(* IEC 61131-3 sources: ae-simplified-sorting-machine/AX/src/packagingSortingMachine, 4 files *)

(* ---- BoxGenerator.st ---- *)
USING SortingMachine;
USING Siemens.Simatic.Crypto;

NAMESPACE SortingMachine

    /// Configuration structure for BoxGenerator
    TYPE
        BoxGeneratorConfig : STRUCT
            /// Default width for generated boxes
            defaultWidth : INT := 50;
            /// Default start position for generated boxes
            defaultStartPosition : INT := 0;
            /// Color code for X-type boxes (typically green)
            colorX : WSTRING := "0xFF21BA84";
            /// Color code for Y-type boxes (typically yellow)
            colorY : WSTRING := "0xFFE8C100";
            /// Starting ID for box numbering (auto-incremented)
            startingId : UINT := UINT#1;
            /// Enable automatic ID increment
            autoIncrementId : BOOL := TRUE;
        END_STRUCT;

    END_TYPE

    /// Box generator class for creating different types of boxes
    /// Provides methods to generate X-type, Y-type, and random boxes with configurable properties
    CLASS PUBLIC BoxGenerator
        VAR PRIVATE
            /// Configuration for the box generator
            _config : BoxGeneratorConfig;
            /// Current ID counter for generated boxes
            _currentId : UINT := UINT#1;
        END_VAR

        /// Constructor to configure the box generator
        METHOD PUBLIC CONSTRUCTOR
            VAR_INPUT
                /// Configuration structure with default values and color settings
                config : BoxGeneratorConfig;
            END_VAR
            _config := config;
            _currentId := _config.startingId;
        END_METHOD

        /// Constructor with individual parameters for convenience
        METHOD PUBLIC CONSTRUCTOR
            VAR_INPUT
                /// Default width for all generated boxes
                defaultWidth : INT;
                /// Default start position for all generated boxes
                defaultStartPosition : INT;
                /// Color code for X-type boxes
                colorX : WSTRING;
                /// Color code for Y-type boxes
                colorY : WSTRING;
                /// Starting ID for box numbering
                startingId : UINT := UINT#1;
            END_VAR
            _config.defaultWidth := defaultWidth;
            _config.defaultStartPosition := defaultStartPosition;
            _config.colorX := colorX;
            _config.colorY := colorY;
            _config.startingId := startingId;
            _config.autoIncrementId := TRUE;
            _currentId := startingId;
        END_METHOD

        /// Create a new box
        METHOD PRIVATE CreateBox
            VAR_INPUT
                /// Optional custom ID, if 0 uses auto-increment
                customId : UINT := UINT#0;
                /// Optional custom start position, if 0 uses default
                customStartPos : INT := 0;
                /// Color to use for the box
                customColor : WSTRING;
            END_VAR
            VAR_IN_OUT
                /// New BasicBox instance configured as specified
                newBox : BasicBox;
            END_VAR

            VAR_TEMP
                useId : UINT;
                useStartPos : INT;
            END_VAR

            // Determine ID to use
            IF customId <> UINT#0 THEN
                useId := customId;
            ELSE
                useId := _currentId;
                IF _config.autoIncrementId THEN
                    _currentId := _currentId + UINT#1;
                END_IF;
            END_IF;

            // Determine start position to use
            IF customStartPos <> 0 THEN
                useStartPos := customStartPos;
            ELSE
                useStartPos := _config.defaultStartPosition;
            END_IF;

            newBox.CONSTRUCT(
                id := useId,
                baseColor := customColor,
                width := _config.defaultWidth,
                startPosition := useStartPos
            );
        END_METHOD

        /// Create a new X-type box (typically green)
        METHOD PUBLIC CreateBoxX
            VAR_INPUT
                /// Optional custom ID, if 0 uses auto-increment
                customId : UINT := UINT#0;
                /// Optional custom start position, if 0 uses default
                customStartPos : INT := 0;
            END_VAR
            VAR_IN_OUT
                /// New BasicBox instance configured as X-type
                newBox : BasicBox;
            END_VAR

            THIS.CreateBox(
                customId := customId,
                customStartPos := customStartPos,
                customColor := _config.colorX,
                newBox := newBox);
        END_METHOD

        /// Create a new Y-type box (typically yellow)
        METHOD PUBLIC CreateBoxY
            VAR_INPUT
                /// Optional custom ID, if 0 uses auto-increment
                customId : UINT := UINT#0;
                /// Optional custom width, if 0 uses default (currently unused)
                customWidth : INT := 0;
                /// Optional custom start position, if 0 uses default
                customStartPos : INT := 0;
            END_VAR
            VAR_IN_OUT
                /// New BasicBox instance configured as Y-type
                newBox : BasicBox;
            END_VAR

            THIS.CreateBox(
                customId := customId,
                customStartPos := customStartPos,
                customColor := _config.colorY,
                newBox := newBox);
        END_METHOD

        /// Create a random box (randomly X-type or Y-type)
        METHOD PUBLIC CreateRandomBox
            VAR_INPUT
                /// Optional custom ID, if 0 uses auto-increment
                customId : UINT := UINT#0;
                /// Optional custom start position, if 0 uses default
                customStartPos : INT := 0;
            END_VAR
            VAR_IN_OUT
                /// New BasicBox instance with random type (X or Y)
                newBox : BasicBox;
            END_VAR
            VAR_TEMP
                randomValue : UDINT;
                useColor : WSTRING;
            END_VAR

            // Generate random value using simple linear congruential generator
            randomValue := Random();

            // Determine color based on random value (even = X, odd = Y)
            IF (randomValue MOD UDINT#2) = UDINT#0 THEN
                useColor := _config.colorX;
            ELSE
                useColor := _config.colorY;
            END_IF;

            THIS.CreateBox(
                customId := customId,
                customStartPos := customStartPos,
                customColor := useColor,
                newBox := newBox);
        END_METHOD

        /// Get the current configuration
        METHOD PUBLIC GetConfig : BoxGeneratorConfig
            GetConfig := _config;
        END_METHOD

        /// Update the configuration
        METHOD PUBLIC SetConfig
            VAR_INPUT
                /// New configuration to apply
                config : BoxGeneratorConfig;
            END_VAR
            _config := config;
        END_METHOD

        /// Get the current ID that would be used for the next box
        METHOD PUBLIC GetCurrentId : UINT
            GetCurrentId := _currentId;
        END_METHOD

        /// Set the current ID counter
        METHOD PUBLIC SetCurrentId
            VAR_INPUT
                /// New ID value to use for subsequent boxes
                newId : UINT;
            END_VAR
            _currentId := newId;
        END_METHOD

        /// Reset the ID counter to the starting value
        METHOD PUBLIC ResetIdCounter
            _currentId := _config.startingId;
        END_METHOD
    END_CLASS

END_NAMESPACE

(* ---- IBasicBox.st ---- *)
NAMESPACE SortingMachine

    /// Data structure representing box properties and status
    /// Used for tracking boxes within the sorting machine system
    INTERFACE IBasicBox
        //=============================================================================
        //SIEMENS AG
        //(c)Copyright 2025 All Rights Reserved
        //-----------------------------------------------------------------------------
        //Tested with:   S7-1500 FW V4.0
        //Engineering:   SIMATIC AX Logic Control Engineering
        //Requirements:  none
        //Functionality: Data structure representing box properties and status
        //-----------------------------------------------------------------------------
        //Change log table:
        //Version  Date       Expert in charge                Changes applied
        //01.00.00 28.11.2025 Siemens Industry Online Support First Release
        //=============================================================================

        /// Constructor to be called once and set private variables
        METHOD CONSTRUCT
            VAR_INPUT
                id : UINT;
                baseColor : WSTRING;
                width   : INT;
                startPosition : INT;
            END_VAR
        END_METHOD

        /// Clear all Data from _boxData
        METHOD  ClearData : BOOL
        END_METHOD

        /// Move the Boxe using the inputed increment value
        METHOD  MoveIncrement : INT
            VAR_INPUT
                increment : INT;
            END_VAR
        END_METHOD

        /// Get Box internal Data
        METHOD  GetBoxData : typeBoxData
        END_METHOD
    END_INTERFACE
END_NAMESPACE

(* ---- AutomaticModeCoordinator.st ---- *)
USING SortingMachine;
USING IEC;
USING Siemens.Simatic.Alarming;

NAMESPACE SortingMachine
    /// Function block for coordinating automatic mode operation of the sorting machine
    /// Handles the automatic flow of boxes through conveyor stations and elevator
    /// Manages the sequence: ConveyorStation1 → Elevator → ConveyorStation2/3 based on box properties
    FUNCTION_BLOCK AutomaticModeCoordinator
        //=============================================================================
        //SIEMENS AG
        //(c)Copyright 2025 All Rights Reserved
        //-----------------------------------------------------------------------------
        //Tested with:   S7-1500 FW V4.0
        //Engineering:   SIMATIC AX Logic Control Engineering
        //Requirements:  none
        //Functionality: Automatic mode coordinator for sorting machine
        //-----------------------------------------------------------------------------
        //Change log table:
        //Version  Date       Expert in charge                Changes applied
        //01.00.00 28.11.2025 Siemens Industry Online Support First Release
        //=============================================================================
        VAR_INPUT
            /// Enable automatic mode operation
            enable : BOOL;
            /// Reset the automatic sequence to initial state
            reset : BOOL;
        END_VAR
        VAR_OUTPUT
            /// Automatic mode is active and running
            active : BOOL;
            /// Error occurred during automatic operation
            error : BOOL;
            /// Status code describing current operation
            status : WORD;
            /// Stored boxes after output conveyors
            storedBoxes : typeStorageInterface;
        END_VAR
        VAR_IN_OUT
            /// Reference to input conveyor station
            conveyorStation1 : ConveyorStation;
            /// Reference to elevator station
            elevatorStation : ElevatorBiStateStation;
            /// Reference to upper output conveyor station
            conveyorStation2 : ConveyorStation;
            /// Reference to lower output conveyor station
            conveyorStation3 : ConveyorStation;
            /// Initial box to use for starting the sequence
            initialBox : BasicBox;
        END_VAR
        VAR PRIVATE
            /// Maximum timeout for operations (30 seconds)
            _maxOperationTime : TIME := T#30s;
            /// Scaner simulation timer to continue
            _scanStationTime : TON;
            /// Elevator delay time for the visualization
            _elevatorDelayTime : TON;
            /// Coordinator was previously reset
            _prevReset : BOOL;
            /// Box amount tracker
            _boxAmountTracker : BoxAmountTracker;
            /// S7-1500 program Alarm for Automatic mode coordenator
            {S7.Alarm = NoAck, "Automatic Mode in Error"}
            alarmAutomaticMode : ProgramAlarm;
        END_VAR
        VAR_TEMP
            elevatorPosition : typeElevatorPosition;
        END_VAR
        VAR CONSTANT
            // Scanner simulation time
            SCAN_SIMULATION_TIME : LTIME := LTIME#2S;
            // Elevator Delay simulation time
            ELEVATOR_SIMULATION_TIME : LTIME := LTIME#1S;
        END_VAR
        // Handle reset request
        IF reset AND NOT _prevReset THEN
            error := FALSE;
            _scanStationTime(IN := FALSE);
            _elevatorDelayTime(IN := FALSE);
            status := typeAutomaticModeCoordinatorStatus#STATUS_RESET_COMPLETE;
        END_IF;
        // Update active status
        active := enable AND NOT error;
        _scanStationTime(IN := conveyorStation1.ReadyToRemoveBox(), PT := SCAN_SIMULATION_TIME);
        _elevatorDelayTime(IN := elevatorStation.ReadyToRemoveBox(), PT := ELEVATOR_SIMULATION_TIME);
        // Update previous flags
        _prevReset := reset;
        // Automatic mode alarm
        alarmAutomaticMode(sig := error);
        // Only run if enabled
        IF NOT (enable OR error) THEN
            status := typeAutomaticModeCoordinatorStatus#STATUS_AUTOMATIC_MODE_DISABLED;
            RETURN;
        END_IF;
        // Check for errors in stations and stop if there are errors
        IF conveyorStation1.GetError()
            OR elevatorStation.GetError()
            OR conveyorStation2.GetError()
            OR conveyorStation3.GetError()
            OR error THEN
            error := TRUE;
            status := typeAutomaticModeCoordinatorStatus#ERR_STATION_FAULT;
            RETURN;
        ELSE
            status := typeAutomaticModeCoordinatorStatus#STATUS_NO_CALL;
        END_IF;

        // Automatic handling for each station
        // Conveyor Station 1:
        // Add initial box if needed
        IF initialBox.BoxData.isPresent AND conveyorStation1.ReadyToReciveBox() THEN
            conveyorStation1.AddNewBox(initialBox);
            initialBox.ClearData();
        // Move box from conv1 to elevator if needed
        ELSIF _scanStationTime.Q AND elevatorStation.ReadyToReciveBox() THEN
            elevatorStation.AddNewBox(conveyorStation1.RemoveBox());
        // Move conveyor boxes
        ELSIF NOT conveyorStation1.GetIsMoving() THEN
                conveyorStation1.MoveIncrementForward();
        END_IF;

        // Elevator 1:
        // Move box from elevator to conveyors
        IF _elevatorDelayTime.Q  OR TRUE THEN
            elevatorPosition := elevatorStation.GetElevatorPositionEnum();
            CASE elevatorPosition OF
                typeElevatorPosition#WORK_POS_1, typeElevatorPosition#HOME:
                    // Transfer to lower output conveyor (ConveyorStation3)
                    IF conveyorStation3.ReadyToReciveBox() THEN
                        conveyorStation3.AddNewBox(elevatorStation.RemoveBox());
                    END_IF;
                typeElevatorPosition#WORK_POS_2:
                    // Transfer to upper output conveyor (ConveyorStation2)
                    IF conveyorStation2.ReadyToReciveBox() THEN
                        conveyorStation2.AddNewBox(elevatorStation.RemoveBox());
                    END_IF;
            END_CASE;
        END_IF;

        // Conveyor 2:
        // Remove boxes from output conveyor 2
        IF conveyorStation2.ReadyToRemoveBox() THEN
            conveyorStation2.RemoveBox();
            _boxAmountTracker.addBoxY := TRUE;
        // Continue moving Conveyor
        ELSIF NOT conveyorStation2.GetIsMoving() THEN
            conveyorStation2.MoveIncrementForward();
        END_IF;
        // Conveyor 3:
        // Remove boxes from output conveyor 3
        IF conveyorStation3.ReadyToRemoveBox() THEN
            conveyorStation3.RemoveBox();
            _boxAmountTracker.addBoxX := TRUE;
        // Continue moving Conveyor
        ELSIF NOT conveyorStation3.GetIsMoving() THEN
            conveyorStation3.MoveIncrementForward();
        END_IF;

        // Track box additions
        _boxAmountTracker(
            reset := reset,
            storedBoxes => storedBoxes);
        // Reset add box inputs for next cycle
        _boxAmountTracker.addBoxX := FALSE;
        _boxAmountTracker.addBoxY := FALSE;

    END_FUNCTION_BLOCK
END_NAMESPACE

(* ---- BasicBox.st ---- *)
NAMESPACE SortingMachine
    /// Basic implementation of a Box in the sorting machine
    CLASS PUBLIC BasicBox IMPLEMENTS IBasicBox
        //=============================================================================
        //SIEMENS AG
        //(c)Copyright 2025 All Rights Reserved
        //-----------------------------------------------------------------------------
        //Tested with:   S7-1500 FW V4.0
        //Engineering:   SIMATIC AX Logic Control Engineering
        //Requirements:  none
        //Functionality: Data structure representing box properties and status
        //-----------------------------------------------------------------------------
        //Change log table:
        //Version  Date       Expert in charge                Changes applied
        //01.00.00 28.11.2025 Siemens Industry Online Support First Release
        //=============================================================================
        VAR PUBLIC
            /// Box data with all relevant properties
            BoxData : typeBoxData;
        END_VAR

        /// Constructor to be called once and set variables
        METHOD PUBLIC CONSTRUCT
            VAR_INPUT
                id : UINT;
                baseColor : WSTRING;
                width   : INT;
                startPosition : INT;
            END_VAR
            BoxData.id := id;
            BoxData.baseColor := baseColor;
            BoxData.isPresent := TRUE;
            BoxData.width := width;
            BoxData.posLeft := startPosition;
            ;
        END_METHOD

        /// Constructor to be called once and set variables based on another Box properties
        METHOD PUBLIC CONSTRUCT
            VAR_IN_OUT
                newBox : BasicBox;
            END_VAR
            BoxData := newBox.BoxData;
            ;
        END_METHOD

        /// Constructor to be called once and set variables based on another Box properties
        METHOD PUBLIC CONSTRUCT
            VAR_INPUT
                newBox : typeBoxData;
            END_VAR
            BoxData := newBox;
            ;
        END_METHOD

        /// Clear all Data from _boxData
        METHOD PUBLIC ClearData : BOOL
            BoxData.id := UINT#0;
            BoxData.stationNr := UINT#0;
            BoxData.isFaulty := FALSE;
            BoxData.baseColor := WSTRING#'';
            BoxData.posLeft := INT#0;
            BoxData.isPresent := FALSE;
            ;
        END_METHOD

        /// Move the Boxe using the inputed increment value
        METHOD PUBLIC MoveIncrement : INT
            VAR_INPUT
                increment : INT;
            END_VAR
            BoxData.posLeft := BoxData.posLeft + increment;
            MoveIncrement := BoxData.posLeft;
        END_METHOD

        /// Get Box internal Data
        /// Only used when data exchanged via Class interface and not using the class itself
        METHOD PUBLIC GetBoxData : typeBoxData
            GetBoxData := BoxData;
        END_METHOD
END_CLASS

END_NAMESPACE
